FUNCTION_BLOCK AxesManager
VAR_INPUT
END_VAR
VAR
	xAchse: AXIS_REF;
	zAchse: AXIS_REF;
	fbMcPowerX: MC_Power;
	fbMcPowerZ: MC_Power;
	fbMcMoveX: MC_MoveAbsolute;
	fbMcMoveZ: MC_MoveAbsolute;
END_VAR

xAchse.ReadStatus();
zAchse.ReadStatus();

METHOD PUBLIC GoTo : BOOL
VAR_INPUT
	stCurPoint: REFERENCE TO ST_2DPoint;
END_VAR
VAR_OUTPUT
	Done: BOOL := FALSE;
END_VAR
fbMcMoveX(
	Axis := xAchse,
	Execute := TRUE,
	Position := stCurPoint.x
);

fbMcMoveZ(
	Axis := zAchse,
	Execute := TRUE,
	Position := stCurPoint.y
);

// Punkt angefahren
Done := fbMcMoveX.Done AND fbMcMoveZ.Done; 

IF Done THEN
	// Bausteine einmal falsen
	fbMcMoveX(Axis := xAchse, Execute := FALSE);
	fbMcMoveZ(Axis := zAchse, Execute := FALSE);
END_IF
END_METHOD

METHOD PUBLIC Init : BOOL
VAR_INPUT
END_VAR
fbMcPowerX(
	Axis := xAchse,
	Enable := TRUE,
	Enable_Positive := TRUE,
	Enable_Negative := TRUE
);

fbMcPowerZ(
	Axis := zAchse,
	Enable := TRUE,
	Enable_Positive := TRUE,
	Enable_Negative := TRUE
);

fbMcPowerX.Status;
END_METHOD

PROPERTY PUBLIC Initialized : BOOL
GET
// Beide Achsen bereit? => TRUE
Initialized := fbMcPowerX.Status AND fbMcPowerZ.Status;
END_GET
END_PROPERTY

METHOD PUBLIC Stop : BOOL
VAR_INPUT
END_VAR
fbMcPowerX(
	Axis := xAchse,
	Enable := FALSE
);

fbMcPowerZ(
	Axis := zAchse,
	Enable := FALSE
);
END_METHOD

PROPERTY PUBLIC Stopped : BOOL
GET
// Beide Achsen gestoppt? => TRUE
Stopped := NOT fbMcPowerX.Status AND NOT fbMcPowerZ.Status;
END_GET
END_PROPERTY

END_FUNCTION_BLOCK

(* stored: Version 1.1.0.1, ProductVersion 3.1.4024.3
   POU AxesManager: Id {7c186c17-78fa-4986-8d65-72678df35783}, SpecialFunc None
   Method GoTo: Id {fff30281-fb10-4a9d-80e7-821a849e41b3}
   Method Init: Id {db33a203-c223-4835-ad49-07c2e911f40d}
   Property Initialized: Id {5c1eb9de-02f5-4dd5-8d7b-713f0c39305a}
   Get Get: Id {c61ad930-fd40-4e46-984f-e961f9efa10a}
   Method Stop: Id {feb14196-459b-441f-8d72-bc125e693eab}
   Property Stopped: Id {48f0ee4d-0b73-471e-96a3-13e20f70b7a5}
   Get Get: Id {480076b0-96f5-412d-9c1a-9a17dad2640a} *)
